// TIA Portal V20 export
VAR_GLOBAL   // PLC tag table "PROFIsafe Drives"
   BA040AZSDR1_Status AT %I5100.0 : "safety.LDrvSafe_typeSinaTlg901Status";
   BA040AZSDR1_Control AT %Q5100.0 : "safety.LDrvSafe_typeSinaTlg901Control";
   BA040AZSDR2_Status AT %I5140.0 : "safety.LDrvSafe_typeSinaTlg901Status";
   BA040AZSDR2_Control AT %Q5140.0 : "safety.LDrvSafe_typeSinaTlg901Control";
   BA040AZSDR3_Status AT %I5180.0 : "safety.LDrvSafe_typeSinaTlg901Status";
   BA040AZSDR3_Control AT %Q5180.0 : "safety.LDrvSafe_typeSinaTlg901Control";
   BA040AZSDR4_Status AT %I5220.0 : "safety.LDrvSafe_typeSinaTlg901Status";
   BA040AZSDR4_Control AT %Q5220.0 : "safety.LDrvSafe_typeSinaTlg901Control";
   BA040AZSDR5_Status AT %I5254.0 : "safety.LDrvSafe_typeSinaTlg901Status";
   BA040AZSDR5_Control AT %Q5254.0 : "safety.LDrvSafe_typeSinaTlg901Control";
   BA040AZSDR6_Status AT %I5288.0 : "safety.LDrvSafe_typeSinaTlg901Status";
   BA040AZSDR6_Control AT %Q5288.0 : "safety.LDrvSafe_typeSinaTlg901Control";
   BA040AZSDR7_Status AT %I5322.0 : "safety.LDrvSafe_typeSinaTlg901Status";
   BA040AZSDR7_Control AT %Q5322.0 : "safety.LDrvSafe_typeSinaTlg901Control";
   BA040AZSDR8_Status AT %I5356.0 : "safety.LDrvSafe_typeSinaTlg901Status";
   BA040AZSDR8_Control AT %Q5356.0 : "safety.LDrvSafe_typeSinaTlg901Control";
   BA040AZSDR9_Status AT %I5390.0 : "safety.LDrvSafe_typeSinaTlg901Status";
   BA040AZSDR9_Control AT %Q5390.0 : "safety.LDrvSafe_typeSinaTlg901Control";
   BA040AZSDR10_Status AT %I5424.0 : "safety.LDrvSafe_typeSinaTlg901Status";
   BA040AZSDR10_Control AT %Q5424.0 : "safety.LDrvSafe_typeSinaTlg901Control";
   BA040AZSDR11_Status AT %I5468.0 : "safety.LDrvSafe_typeSinaTlg901Status";
   BA040AZSDR11_Control AT %Q5468.0 : "safety.LDrvSafe_typeSinaTlg901Control";
   BA040AZSDR12_Status AT %I5502.0 : "safety.LDrvSafe_typeSinaTlg901Status";
   BA040AZSDR12_Control AT %Q5502.0 : "safety.LDrvSafe_typeSinaTlg901Control";
   BA040AZSDR13_Status AT %I5546.0 : "safety.LDrvSafe_typeSinaTlg901Status";
   BA040AZSDR13_Control AT %Q5546.0 : "safety.LDrvSafe_typeSinaTlg901Control";
   BA040AZSDR14_Status AT %I5590.0 : "safety.LDrvSafe_typeSinaTlg901Status";
   BA040AZSDR14_Control AT %Q5590.0 : "safety.LDrvSafe_typeSinaTlg901Control";
   BA040AZSDR15_Status AT %I5634.0 : "safety.LDrvSafe_typeSinaTlg901Status";
   BA040AZSDR15_Control AT %Q5634.0 : "safety.LDrvSafe_typeSinaTlg901Control";
   BA040AZSDR16_Status AT %I5668.0 : "safety.LDrvSafe_typeSinaTlg901Status";
   BA040AZSDR16_Control AT %Q5668.0 : "safety.LDrvSafe_typeSinaTlg901Control";
   BA040AZSDR17_Status AT %I5702.0 : "safety.LDrvSafe_typeSinaTlg901Status";
   BA040AZSDR17_Control AT %Q5702.0 : "safety.LDrvSafe_typeSinaTlg901Control";
   BA040AZSDR18_Status AT %I5736.0 : "safety.LDrvSafe_typeSinaTlg901Status";
   BA040AZSDR18_Control AT %Q5736.0 : "safety.LDrvSafe_typeSinaTlg901Control";
   BA040AZSDR19_Status AT %I5770.0 : "safety.LDrvSafe_typeSinaTlg901Status";
   BA040AZSDR19_Control AT %Q5770.0 : "safety.LDrvSafe_typeSinaTlg901Control";
   BA040AZSDR20_Status AT %I5804.0 : "safety.LDrvSafe_typeSinaTlg901Status";
   BA040AZSDR20_Control AT %Q5804.0 : "safety.LDrvSafe_typeSinaTlg901Control";
   BA040AZSDR21_Status AT %I5838.0 : "safety.LDrvSafe_typeSinaTlg901Status";
   BA040AZSDR21_Control AT %Q5838.0 : "safety.LDrvSafe_typeSinaTlg901Control";
   BA040AZSDR22_Status AT %I5872.0 : "safety.LDrvSafe_typeSinaTlg901Status";
   BA040AZSDR22_Control AT %Q5872.0 : "safety.LDrvSafe_typeSinaTlg901Control";
   BA040AZSDR23_Status AT %I5906.0 : "safety.LDrvSafe_typeSinaTlg901Status";
   BA040AZSDR23_Control AT %Q5906.0 : "safety.LDrvSafe_typeSinaTlg901Control";
   BA040AZSDR24_Status AT %I5940.0 : "safety.LDrvSafe_typeSinaTlg901Status";
   BA040AZSDR24_Control AT %Q5940.0 : "safety.LDrvSafe_typeSinaTlg901Control";
   BA040AZSDR25_Status AT %I5984.0 : "safety.LDrvSafe_typeSinaTlg901Status";
   BA040AZSDR25_Control AT %Q5984.0 : "safety.LDrvSafe_typeSinaTlg901Control";
   BA040AZSDR26_Status AT %I6018.0 : "safety.LDrvSafe_typeSinaTlg901Status";
   BA040AZSDR26_Control AT %Q6018.0 : "safety.LDrvSafe_typeSinaTlg901Control";
   BA040AZSDR27_Status AT %I6062.0 : "safety.LDrvSafe_typeSinaTlg901Status";
   BA040AZSDR27_Control AT %Q6062.0 : "safety.LDrvSafe_typeSinaTlg901Control";
   BA040AZSDR28_Status AT %I6096.0 : "safety.LDrvSafe_typeSinaTlg901Status";
   BA040AZSDR28_Control AT %Q6096.0 : "safety.LDrvSafe_typeSinaTlg901Control";
   BA040AZSDR29_Status AT %I6140.0 : "safety.LDrvSafe_typeSinaTlg901Status";
   BA040AZSDR29_Control AT %Q6140.0 : "safety.LDrvSafe_typeSinaTlg901Control";
   BA040AZSDR30_Status AT %I6174.0 : "safety.LDrvSafe_typeSinaTlg901Status";
   BA040AZSDR30_Control AT %Q6174.0 : "safety.LDrvSafe_typeSinaTlg901Control";
   BA040AZSDR31_Status AT %I6218.0 : "safety.LDrvSafe_typeSinaTlg901Status";
   BA040AZSDR31_Control AT %Q6218.0 : "safety.LDrvSafe_typeSinaTlg901Control";
   BA040AZSDR32_Status AT %I6262.0 : "safety.LDrvSafe_typeSinaTlg901Status";
   BA040AZSDR32_Control AT %Q6262.0 : "safety.LDrvSafe_typeSinaTlg901Control";
   BA040AZSDR33_Status AT %I6306.0 : "safety.LDrvSafe_typeSinaTlg901Status";
   BA040AZSDR33_Control AT %Q6306.0 : "safety.LDrvSafe_typeSinaTlg901Control";
   BA040AZSDR34_Status AT %I6350.0 : "safety.LDrvSafe_typeSinaTlg901Status";
   BA040AZSDR34_Control AT %Q6350.0 : "safety.LDrvSafe_typeSinaTlg901Control";
   BA040AZSDR35_Status AT %I6384.0 : "safety.LDrvSafe_typeSinaTlg901Status";
   BA040AZSDR35_Control AT %Q6384.0 : "safety.LDrvSafe_typeSinaTlg901Control";
   BA040AZSDR36_Status AT %I6428.0 : "safety.LDrvSafe_typeSinaTlg901Status";
   BA040AZSDR36_Control AT %Q6428.0 : "safety.LDrvSafe_typeSinaTlg901Control";
   BA040AZSDR37_Status AT %I6462.0 : "safety.LDrvSafe_typeSinaTlg901Status";
   BA040AZSDR37_Control AT %Q6462.0 : "safety.LDrvSafe_typeSinaTlg901Control";
   BA040AZSDR38_Status AT %I6506.0 : "safety.LDrvSafe_typeSinaTlg901Status";
   BA040AZSDR38_Control AT %Q6506.0 : "safety.LDrvSafe_typeSinaTlg901Control";
   BA040AZSDR39_Status AT %I6540.0 : "safety.LDrvSafe_typeSinaTlg901Status";
   BA040AZSDR39_Control AT %Q6540.0 : "safety.LDrvSafe_typeSinaTlg901Control";
   BA040AZSDR40_Status AT %I6574.0 : "safety.LDrvSafe_typeSinaTlg901Status";
   BA040AZSDR40_Control AT %Q6574.0 : "safety.LDrvSafe_typeSinaTlg901Control";
   BA040AZSDR41_Status AT %I6608.0 : "safety.LDrvSafe_typeSinaTlg901Status";
   BA040AZSDR41_Control AT %Q6608.0 : "safety.LDrvSafe_typeSinaTlg901Control";
END_VAR
